FUNCTION_BLOCK BLOCK_CLIGNOTANT
VAR_INPUT
	PRM_PERIOD:	TIME;
END_VAR
VAR_OUTPUT
	STATE: 		BOOL;
END_VAR
VAR
	TIMER_ON:	TP;
	TIMER_OFF:	TP;
END_VAR

TIMER_ON(IN:=NOT TIMER_OFF.Q ,PT:= PRM_PERIOD);
TIMER_OFF(IN:=NOT TIMER_ON.Q,PT:=PRM_PERIOD);
STATE := TIMER_ON.Q;

END_FUNCTION_BLOCK

(* stored: Version 1.1.0.1, ProductVersion 3.1.4024.10
   POU BLOCK_CLIGNOTANT: Id {feb5943c-c1ba-4f2d-9054-011dbdc85015}, SpecialFunc None *)
